FUNCTION_BLOCK FB_ShippingHoming EXTENDS FB_ActionBasic
VAR_INPUT
	xExecute 	: BOOL;
	xAbort 		: BOOL;
    FanucRobot 	: REFERENCE TO FB_FanucRobot_Basic_V2;
	Homed 		: REFERENCE TO BOOL;
	input		: REFERENCE TO ST_InputTable;
	Service		: REFERENCE TO ST_ShippingService;
	Motor		: REFERENCE TO UNI_MotorList;
END_VAR
VAR_OUTPUT
	xAborted : BOOL;
	iErrorID : INT;
	ErrorMsg : STRING;
	RobotResetCMD : BOOL;
END_VAR
VAR
	StateBehaviour 		 : CBML.ETrigA;
	uiShippingHomingStep : UINT;
	FanucRobotCheckTon 	 	: TON;
	ResetRobotDelay 	 	: TON;
	TON_RobotFeedOutCommand : TON;
	TON_RobotTimeOut		: TON;
	fbExecuteEdgeDetect  :FB_EdgeDetect;
	_fbShippingRobot_TransmitCVEnd	: FB_ShippingRobot_TransmitCVEnd;
	TON_RobotRSR01_Delay	: TON;
END_VAR

A00_BasicUnits();
THIS^.IBehaviourModel := StateBehaviour;
StateBehaviour(xExecute := xExecute,
    xDone => xDone,
    xBusy => xBusy,
    xError => xError,
    xAbort := xAbort OR fbExecuteEdgeDetect.xFallingEdge,
    xAborted => xAborted);

//Error Msg
iErrorID := StateBehaviour._model.iErrorID;
ErrorMsg := M_GetErrorMsg(xErrorID := iErrorID);


//Make sure that C# turns off execute to shut down the service
fbExecuteEdgeDetect(xInput :=xExecute);

ACTION A00_BasicUnits:
FanucRobotCheckTon(PT := T#90S);		//All Service TimeOut
ResetRobotDelay(PT:=T#300MS);
TON_RobotFeedOutCommand(PT:= T#5S);		//Robot FeedOut Command TimeOut
TON_RobotTimeOut(PT := T#60S);			//Robot FeedOut Service Done Time
TON_RobotRSR01_Delay(PT :=T#3S);

_fbShippingRobot_TransmitCVEnd(
	Execute:= , 
	Abort:= , 
	Reset:= , 
	ObjectName:= , 
	Busy=> , 
	Done=> , 
	Aborted=> , 
	Error=> , 
	ErrorID=> , 
	Status=> , 
	UniqueErrorCode=> , 
	Robot:= fanucrobot, 
	Info:= , 
	Stop:= , 
	INPUT:= input, 
	Motor:= Motor, 
	bCompleteRequest:= ,
	fbSHippingHomingBusy := THIS^.xBusy);
END_ACTION

METHOD CleanupAction
VAR_INPUT
    xAbortProposed : BOOL;
    iErrorIDProposed: INT;
END_VAR
VAR_OUTPUT
    xComplete : BOOL := TRUE;
    xAbort: BOOL := xAbortProposed;
 	iErrorID : INT := iErrorIDProposed;
END_VAR
RobotResetCMD := FALSE;
FanucRobotCheckTon.IN := FALSE;
uiShippingHomingStep := 0;
END_METHOD

METHOD CyclicAction
VAR_INPUT
    itfTimingController : CBML.ITimingController;
END_VAR
VAR_OUTPUT
    xComplete : BOOL := TRUE;
    iErrorID : INT := 0;
END_VAR
xComplete := FALSE;
CASE uiShippingHomingStep OF
	
	0:
			TON_RobotFeedOutCommand.IN  := FALSE;
			TON_RobotTimeOut.IN 		:= FALSE;
			FanucRobotCheckTon.IN 		:= TRUE;
			IF FanucRobot.Error THEN
				RobotResetCMD := TRUE;
				ResetRobotDelay.IN:=TRUE;
			ELSE
				uiShippingHomingStep := 500;
			END_IF
			IF ResetRobotDelay.Q THEN
				ResetRobotDelay.IN :=FALSE;
				uiShippingHomingStep := 500;
			END_IF
		
		
	500:	// 手臂 RSR02 回原點
			ResetRobotDelay.IN := FALSE;
			RobotResetCMD := FALSE;
			FanucRobot.OpMode := E_FanucRobotOpMode.RSR02;
			IF FanucRobot.Error THEN
				RobotResetCMD := TRUE;		
			END_IF
			IF FanucRobot._RSR2_Completed THEN
				uiShippingHomingStep := 600;
			END_IF
			
	600:	// 回完回點後切換為 RSR01 工作模式
			FanucRobot.OpMode := E_FanucRobotOpMode.RSR01;
			IF FanucRobot._RSR1_Ready THEN
				uiShippingHomingStep := 1000;
			END_IF
		
	1000:	// 確認手臂切換到 RSR01 模式，並且確保已回報 PLC 正在執行 RSR01
			IF FanucRobot.OpMode = E_FanucRobotOpMode.RSR01 AND 
				NOT FanucRobot._DI1.Done AND 
				FanucRobot._DI12.RSR1_Active 
			THEN
				uiShippingHomingStep := 1200;
			END_IF
			
	1200:	// 檢查手臂夾具的開合狀態
			TON_RobotRSR01_Delay.IN := FALSE;
			IF NOT fanucRobot._DI1.ClampA_Open THEN
				uiShippingHomingStep := 2000;
			ELSE
				uiShippingHomingStep := 9000;
			END_IF
			
	2000:	// 同尺寸軌道 busy Check
			TON_RobotFeedOutCommand.IN := TRUE;
			_fbShippingRobot_TransmitCVEnd.M_StartHomingFeedOut(UseA := TRUE);
			IF _fbShippingRobot_TransmitCVEnd.Busy THEN
				uiShippingHomingStep := 2100;
			END_IF
			IF TON_RobotFeedOutCommand.Q THEN
				iErrorID := 10;
			END_IF
	
	2100:	// 同尺寸軌道 done Check
			TON_RobotFeedOutCommand.IN := FALSE;
			TON_RobotTimeOut.IN := TRUE;
			IF _fbShippingRobot_TransmitCVEnd.Done THEN
				_fbShippingRobot_TransmitCVEnd.M_ResetHomingFeedOut();		
				uiShippingHomingStep := 0;
			END_IF
			IF TON_RobotTimeOut.Q THEN
				iErrorID := 11;
			END_IF

	9000:	// process done
			FanucRobotCheckTon.IN := FALSE;
			Homed := TRUE;
			xComplete := TRUE;
END_CASE

IF FanucRobotCheckTon.Q THEN
	iErrorID := 4;
END_IF
END_METHOD

METHOD ExitAction
VAR_INPUT
    xAfterCleanup : BOOL;
    xInCopyCode : BOOL;
END_VAR
END_METHOD

METHOD M_GetErrorMsg : T_MaxString
VAR_INPUT
	xErrorID: INT;
END_VAR

VAR
	
END_VAR
CASE xErrorID OF
    0:
        M_GetErrorMsg := 'No Error';
    1:
        M_GetErrorMsg := 'Action time out';
    2:
        M_GetErrorMsg := 'Cylinder not ready';
    3:
        M_GetErrorMsg := 'Motor not ready';
    4:
		M_GetErrorMsg := 'FanucRobot can not homing';
	10:
		M_GetErrorMsg := 'Shipping FanucRobot FeedOut to SameSizeConveyor not busy';
	11:
		M_GetErrorMsg := 'Shipping FanucRobot FeedOut to SameSizeConveyor Done Timeout';
	20:
		M_GetErrorMsg := 'Occupid , AutoMode_ShippingRobot_TransmitCVEnd in Executing ';
END_CASE
END_METHOD

METHOD ResetAction
VAR_OUTPUT
    xComplete : BOOL := TRUE;
END_VAR
FanucRobotCheckTon.IN := FALSE;
TON_RobotRSR01_Delay.IN	:= FALSE;
_fbShippingRobot_TransmitCVEnd.M_ResetHomingFeedOut();
END_METHOD

METHOD StartAction
VAR_OUTPUT
    xComplete : BOOL := TRUE;
	iErrorID : INT := 0;
END_VAR
Homed := FALSE;
FanucRobotCheckTon.IN 		:= FALSE;
ResetRobotDelay.IN 			:= FALSE;
TON_RobotFeedOutCommand.IN 	:= FALSE;
TON_RobotTimeOut.IN 		:= FALSE;
TON_RobotRSR01_Delay.IN		:= FALSE;
uiShippingHomingStep := 0;
_fbShippingRobot_TransmitCVEnd.M_ResetHomingFeedOut();

IF  Service.AutoMode_ShippingRobot_TransmitCVEnd.Command.Execute AND
	Service.AutoMode_ShippingRobot_TransmitCVEnd.Status.Busy AND
	Service.AutoMode_ShippingRobot_TransmitCVEnd.Status.Error 
THEN
	iErrorID := 20;
END_IF
END_METHOD

END_FUNCTION_BLOCK

(* stored: Version 1.1.0.1, ProductVersion 3.1.4024.13
   POU FB_ShippingHoming: Id {fb6a1860-c382-494a-99f6-2de10876296e}, SpecialFunc None
   Folder STATE: Id {4b925b5e-f789-4880-9d0a-0db60304a629}
   Action A00_BasicUnits: Id {f3e17531-2194-49d0-addb-559149d6847b}
   Method CleanupAction: Id {f4a4a7bd-b035-4c68-8efe-6ad0c9c5f25b}
   Method CyclicAction: Id {ccbe0fb7-3c8a-435f-b091-6473cfa1a63d}
   Method ExitAction: Id {b40aaad3-b319-49ad-ab2a-b5db16cceaaa}
   Method M_GetErrorMsg: Id {03eac412-96d4-4e84-bf40-8d06670d8278}
   Method ResetAction: Id {a5d6e6fc-9b41-4dd3-92ef-8e0382f51f5a}
   Method StartAction: Id {a77f2f89-4696-4442-828d-0460ba5f894c} *)
